{attribute 'pack_mode' := '2'}
TYPE ST_GEAR_IN :
STRUCT
  bAdvancedSlaveDynamics  : BOOL;
  nMultiMasterSyncMode    : INT;

  nAxisIndexMaster    : ARRAY [1..4] OF BYTE; // Index of Master1-4
  rGearRatio          : ARRAY [1..4] OF REAL; 
  Acceleration        : REAL;
  Deceleration        : REAL;
  Jerk                : REAL;  
END_STRUCT
END_TYPE

(* stored: Version 1.1.0.1, ProductVersion 3.1.4024.12
   DUT ST_GEAR_IN: Id {4efdd300-d04e-0b13-188d-d85306bab98e} *)
